FUNCTION_BLOCK CMP_P1 (* Composite Function Block Type *)
  (* Standard: 61499-2 *)
  (* Version 0.0, 2015-11-23, 4DIAC-IDE, 4DIAC-Consortium *)
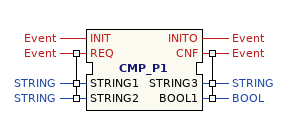
  EVENT_INPUT
    INIT; (* Initialization Request *)
    REQ WITH STRING1, STRING2; (* Normal Execution Request *)
  END_EVENT
  EVENT_OUTPUT
    INITO; (* Initialization Confirm *)
    CNF WITH STRING3, BOOL1; (* Execution Confirmation *)
  END_EVENT
  VAR_INPUT
    STRING1 : STRING;
    STRING2 : STRING;
  END_VAR
  VAR_OUTPUT
    STRING3 : STRING;
    BOOL1 : BOOL;
  END_VAR
  FBS
    E_SPLIT_1_1_0_1_0_0 : E_SPLIT;
    E_SPLIT_1_0_0_0_0_0 : E_SPLIT;
    F_NOT_1_1 : F_NOT;
    STRING2STRING_1ok : STRING2STRING(IN := okk);
    STRING_SPLIT_0_1 : STRING_SPLIT;
    SIFB_RAWSTRING_EQ_0_0_0_0 : SIFB_RAWSTRING_EQ;
    E_SPLIT_1_0_0_0_0 : E_SPLIT;
    E_MERGE_4_0 : E_MERGE;
    E_PERMIT_1_1_0_2 : E_PERMIT;
    E_MERGE_1_0_0 : E_MERGE;
    E_PERMIT_1_1_0_0_1_0 : E_PERMIT;
    CLIENT_1_0_0 : CLIENT_1(QI := BOOL#1, ID := ser[COM3]);
    F_LE_0_0_0 : F_LE(IN2 := UINT#2);
    BASIC_SEND_ENQ_1_0_1 : BASIC_SEND_ENQ;
    STRING_SPLIT_0_0_0 : STRING_SPLIT;
    BASIC_SEND_EOT_0 : BASIC_SEND_EOT;
    E_MERGE_4 : E_MERGE;
    F_NOT_1_0_0_0_0 : F_NOT;
    STRING2STRING_1_1_0_0 : STRING2STRING;
    E_SPLIT_1_1_0_2 : E_SPLIT;
    E_PERMIT_1_1_0_0_0_1_0 : E_PERMIT;
    E_PERMIT_1_0_1_1 : E_PERMIT;
    E_PERMIT_1_1_0_0_0_1_0_0 : E_PERMIT;
    E_PERMIT_1_3_0_0 : E_PERMIT;
    E_SPLIT_1_0_1_0 : E_SPLIT;
    E_PERMIT_1_1_0_0_2 : E_PERMIT;
    SIFB_GENTXT_0 : SIFB_GENTXT;
    E_PERMIT_1_1_0_0_0_1 : E_PERMIT;
    E_MERGE_0_0 : E_MERGE;
    E_DELAY_0_1 : E_DELAY(DT := T#3s);
    F_LE_0_1 : F_LE(IN2 := UINT#2);
    F_NOT_1_0_2 : F_NOT;
    E_SPLIT_1_1_1 : E_SPLIT;
    STRING2STRING_5 : STRING2STRING;
    E_SPLIT_1_1_0_1_1 : E_SPLIT;
    E_SPLIT_1_0_1_1 : E_SPLIT;
    SIFB_RAWSTRING_EQ_0_0_1 : SIFB_RAWSTRING_EQ;
    STRING2STRING_1_1_0_0_0 : STRING2STRING;
    F_NOT_1_0_0_0 : F_NOT;
    E_CTU_0_0_0 : E_CTU(PV := 0);
    E_MERGE_2_2_0 : E_MERGE;
    E_DELAY_0_1_0 : E_DELAY(DT := T#150ms);
    E_SR_2 : E_SR;
    E_CTU_0_1 : E_CTU(PV := 0);
    E_SPLIT_1_0_0_1_0 : E_SPLIT;
    F_NOT_1_0_1_0 : F_NOT;
    E_PERMIT_1_0_1_0_0 : E_PERMIT;
    E_SPLIT_1_0_0_1 : E_SPLIT;
    E_PERMIT_1_3_1 : E_PERMIT;
    E_PERMIT_2 : E_PERMIT;
    BASIC_SEND_NAKDEL_1 : BASIC_SEND_NAKDEL;
    SIFB_SPSTRINGCMP_1 : SIFB_SPSTRINGCMP;
    B_DEMUX_BOOL : B_DEMUX_BOOL(IN2 := BOOL#FALSE, IN3 := BOOL#TRUE);
  END_FBS
  EVENT_CONNECTIONS
    E_SPLIT_1_1_0_1_0_0.EO2 TO E_PERMIT_1_0_1_0_0.EI;
    E_CTU_0_1.CUO TO F_LE_0_1.REQ;
    F_NOT_1_0_2.CNF TO E_SPLIT_1_1_0_1_0_0.EI;
    E_PERMIT_1_1_0_2.EO TO E_SPLIT_1_1_0_2.EI;
    BASIC_SEND_ENQ_1_0_1.EO TO STRING_SPLIT_0_1.EI2;
    E_MERGE_0_0.EO TO BASIC_SEND_EOT_0.REQ;
    E_PERMIT_1_0_1_1.EO TO E_MERGE_0_0.EI1;
    BASIC_SEND_NAKDEL_1.CNF TO SIFB_RAWSTRING_EQ_0_0_0_0.EI;
    E_SPLIT_1_0_0_0_0_0.EO1 TO E_MERGE_4_0.EI2;
    E_CTU_0_1.RO TO E_MERGE_4.EI1;
    STRING2STRING_1ok.CNF TO E_SPLIT_1_0_0_1.EI;
    F_NOT_1_0_0_0_0.CNF TO E_PERMIT_1_1_0_0_0_1_0_0.EI;
    F_NOT_1_0_1_0.CNF TO E_PERMIT_1_1_0_0_1_0.EI;
    E_SPLIT_1_1_1.EO2 TO E_PERMIT_1_1_0_0_2.EI;
    F_LE_0_0_0.CNF TO F_NOT_1_0_2.REQ;
    E_DELAY_0_1_0.EO TO E_SPLIT_1_0_0_0_0_0.EI;
    E_SPLIT_1_1_1.EO3 TO F_NOT_1_0_0_0.REQ;
    CLIENT_1_0_0.CNF TO E_SPLIT_1_0_1_1.EI;
    E_SPLIT_1_0_1_1.EO2 TO E_PERMIT_2.EI;
    E_MERGE_4_0.EO TO E_SR_2.R;
    E_SPLIT_1_1_0_1_1.EO1 TO E_CTU_0_0_0.CU;
    E_SPLIT_1_0_0_0_0_0.EO2 TO E_MERGE_2_2_0.EI1;
    E_SR_2.EO TO E_SPLIT_1_0_0_1_0.EI;
    E_MERGE_1_0_0.EO TO E_CTU_0_1.CU;
    E_PERMIT_2.EO TO STRING_SPLIT_0_0_0.EI1;
    F_NOT_1_1.CNF TO E_PERMIT_1_0_1_1.EI;
    E_SPLIT_1_0_1_0.EO2 TO CLIENT_1_0_0.REQ;
    E_SPLIT_1_1_0_1_0_0.EO1 TO E_PERMIT_1_3_0_0.EI;
    E_SPLIT_1_1_0_2.EO2 TO E_CTU_0_0_0.R;
    STRING2STRING_1_1_0_0.CNF TO STRING2STRING_1_1_0_0_0.REQ;
    STRING_SPLIT_0_0_0.EO TO SIFB_RAWSTRING_EQ_0_0_1.EI;
    E_SPLIT_1_0_1_1.EO3 TO SIFB_GENTXT_0.REQ;
    E_SPLIT_1_0_0_1_0.EO2 TO E_PERMIT_1_1_0_0_0_1_0.EI;
    E_MERGE_4.EO TO STRING2STRING_5.REQ;
    E_SPLIT_1_0_0_1_0.EO1 TO F_NOT_1_0_0_0_0.REQ;
    E_PERMIT_1_1_0_0_1_0.EO TO E_MERGE_1_0_0.EI1;
    E_SPLIT_1_0_1_0.EO1 TO E_DELAY_0_1.START;
    E_SPLIT_1_0_0_1.EO1 TO E_MERGE_4_0.EI1;
    E_PERMIT_1_0_1_0_0.EO TO E_MERGE_0_0.EI2;
    STRING2STRING_5.CNF TO STRING_SPLIT_0_1.EI1;
    STRING_SPLIT_0_1.EO TO E_SPLIT_1_0_1_0.EI;
    BASIC_SEND_EOT_0.CNF TO E_SPLIT_1_0_0_0_0.EI;
    E_PERMIT_1_3_0_0.EO TO E_MERGE_4.EI2;
    E_PERMIT_1_1_0_0_2.EO TO E_SPLIT_1_1_0_1_1.EI;
    E_PERMIT_1_1_0_0_0_1_0_0.EO TO E_MERGE_2_2_0.EI1;
    F_NOT_1_0_0_0.CNF TO E_PERMIT_1_1_0_0_0_1.EI;
    E_DELAY_0_1.EO TO E_MERGE_1_0_0.EI2;
    SIFB_RAWSTRING_EQ_0_0_0_0.EO TO E_SPLIT_1_1_1.EI;
    E_SPLIT_1_0_0_0_0.EO2 TO STRING_SPLIT_0_1.EI3;
    E_SPLIT_1_1_0_2.EO3 TO STRING2STRING_1ok.REQ;
    E_MERGE_2_2_0.EO TO E_DELAY_0_1.STOP;
    F_LE_0_1.CNF TO E_PERMIT_1_3_1.EI;
    SIFB_RAWSTRING_EQ_0_0_1.EO TO BASIC_SEND_NAKDEL_1.REQ;
    E_SPLIT_1_0_0_0_0.EO1 TO E_DELAY_0_1_0.START;
    STRING2STRING_1_1_0_0_0.CNF TO E_SR_2.S;
    F_LE_0_1.CNF TO F_NOT_1_1.REQ;
    E_PERMIT_1_1_0_0_0_1_0.EO TO E_CTU_0_1.R;
    E_SPLIT_1_1_1.EO1 TO E_PERMIT_1_1_0_2.EI;
    E_CTU_0_0_0.CUO TO F_LE_0_0_0.REQ;
    E_PERMIT_1_1_0_0_0_1.EO TO F_NOT_1_0_1_0.REQ;
    E_SPLIT_1_0_1_1.EO1 TO E_MERGE_2_2_0.EI2;
    E_PERMIT_1_3_1.EO TO BASIC_SEND_ENQ_1_0_1.EI;
    INIT TO CLIENT_1_0_0.INIT;
    CLIENT_1_0_0.INITO TO INITO;
    REQ TO STRING2STRING_1_1_0_0.REQ;
    E_SPLIT_1_0_0_1.EO2 TO CNF;
    E_SPLIT_1_0_1_0.EO3 TO SIFB_SPSTRINGCMP_1.EI;
    SIFB_SPSTRINGCMP_1.EO1 TO E_SPLIT_1_1_0_2.EI;
    SIFB_RAWSTRING_EQ_0_0_1.EO TO B_DEMUX_BOOL.EI1;
    SIFB_SPSTRINGCMP_1.EO1 TO B_DEMUX_BOOL.EI3;
    E_SPLIT_1_0_0_0_0.EO3 TO B_DEMUX_BOOL.EI2;
  END_CONNECTIONS
  DATA_CONNECTIONS
    F_NOT_1_1.OUT TO E_PERMIT_1_0_1_1.PERMIT;
    F_NOT_1_0_2.OUT TO E_PERMIT_1_0_1_0_0.PERMIT;
    SIFB_RAWSTRING_EQ_0_0_1.OUT TO E_PERMIT_1_1_0_2.PERMIT;
    E_SR_2.Q TO E_PERMIT_1_1_0_0_0_1_0.PERMIT;
    F_LE_0_0_0.OUT TO E_PERMIT_1_3_0_0.PERMIT;
    SIFB_RAWSTRING_EQ_0_0_0_0.OUT TO E_PERMIT_1_1_0_0_2.PERMIT;
    E_SR_2.Q TO E_PERMIT_2.PERMIT;
    CLIENT_1_0_0.RD_1 TO STRING_SPLIT_0_0_0.STRING1;
    E_SR_2.Q TO F_NOT_1_0_0_0_0.IN;
    CLIENT_1_0_0.RD_1 TO SIFB_GENTXT_0.STRING2;
    SIFB_RAWSTRING_EQ_0_0_0_0.OUT TO F_NOT_1_0_0_0.IN;
    BASIC_SEND_ENQ_1_0_1.OUT TO STRING_SPLIT_0_1.STRING2;
    BASIC_SEND_EOT_0.OUT TO STRING_SPLIT_0_1.STRING3;
    F_LE_0_1.OUT TO F_NOT_1_1.IN;
    F_LE_0_0_0.OUT TO F_NOT_1_0_2.IN;
    STRING_SPLIT_0_0_0.OUT TO SIFB_RAWSTRING_EQ_0_0_0_0.IN1;
    F_NOT_1_0_0_0.OUT TO E_PERMIT_1_1_0_0_0_1.PERMIT;
    BASIC_SEND_NAKDEL_1.OUT TO SIFB_RAWSTRING_EQ_0_0_0_0.IN2;
    E_CTU_0_1.CV TO F_LE_0_1.IN1;
    STRING2STRING_1_1_0_0.OUT TO STRING2STRING_5.IN;
    STRING2STRING_5.OUT TO STRING_SPLIT_0_1.STRING1;
    E_CTU_0_0_0.CV TO F_LE_0_0_0.IN1;
    STRING_SPLIT_0_1.OUT TO CLIENT_1_0_0.SD_1;
    F_NOT_1_0_0_0_0.OUT TO E_PERMIT_1_1_0_0_0_1_0_0.PERMIT;
    F_LE_0_1.OUT TO E_PERMIT_1_3_1.PERMIT;
    F_NOT_1_0_1_0.OUT TO E_PERMIT_1_1_0_0_1_0.PERMIT;
    STRING2STRING_1_1_0_0_0.OUT TO SIFB_RAWSTRING_EQ_0_0_1.IN2;
    STRING_SPLIT_0_0_0.OUT TO SIFB_RAWSTRING_EQ_0_0_1.IN1;
    SIFB_RAWSTRING_EQ_0_0_1.OUT TO F_NOT_1_0_1_0.IN;
    STRING_SPLIT_0_1.OUT TO SIFB_GENTXT_0.STRING1;
    STRING1 TO STRING2STRING_1_1_0_0.IN;
    STRING2 TO STRING2STRING_1_1_0_0_0.IN;
    STRING_SPLIT_0_0_0.OUT TO STRING3;
    STRING2STRING_1_1_0_0_0.OUT TO SIFB_SPSTRINGCMP_1.STRING1;
    SIFB_RAWSTRING_EQ_0_0_1.OUT TO B_DEMUX_BOOL.IN1;
    B_DEMUX_BOOL.OUT TO BOOL1;
  END_CONNECTIONS
END_FUNCTION_BLOCK
